screen "LLCCA_PID" 1280x800, template "Template_main"
   Button "Button_1" at 1170,125 size 106x32; TextOff 'LLCCA_PID / -'
   IOField "I/O field_4" at 220,550 size 66x32; FormatPattern 99.99; Unit  
      ProcessValue <- "LLCCA_PvSim_LLCCA_PID_DB_ioAddFactor"
   TextField "Text field_22" at 220,525 size 59x23; Text 'factor / faktor'
   IOField "I/O field_15" at 290,550 size 61x32; FormatPattern 99; Unit  s 
      ProcessValue <- "LLCCA_PvSim_LLCCA_PID_DB_ioAddTimeLag"
   TextField "Text field_23" at 290,525 size 45x23; Text 'tLag'
   Button "Button_4" at 220,680 size 156x32; TextOff 'Reset / Återställning'
      on Release: SetBit("RUN_DB_resetPvSim")
   IOField "I/O field_21" at 355,550 size 61x32; FormatPattern 999; Unit  s 
      ProcessValue <- "LLCCA_PvSim_LLCCA_PID_DB_ioAddFilter"
   TextField "Text field_25" at 355,525 size 51x23; Text 'filter'
   IOField "I/O field_22" at 220,615 size 66x32; FormatPattern 99.99; Unit  
      ProcessValue <- "LLCCA_PvSim_LLCCA_PID_DB_ioSubFactor"
   TextField "Text field_26" at 220,590 size 59x23; Text 'factor / faktor'
   IOField "I/O field_23" at 420,615 size 96x32; FormatPattern 99.9; Unit   U 
      ProcessValue <- "LLCCA_PvSim_LLCCA_PID_DB_ioSubStartValue"
   TextField "Text field_27" at 420,590 size 104x23; Text 'start value / omgivningstemp.'
   TextField "Text field_28" at 10,525 size 186x23; Text 'Additive component / Värmning'
   TextField "Text field_29" at 10,590 size 213x23; Text 'subtracting component / Kylning'
   IOField "I/O field_16" at 10,550 size 161x32; FormatPattern 999.9; Unit  U/min 
      ProcessValue <- "LLCCA_PvSim_LLCCA_PID_DB_addComp"
   IOField "I/O field_17" at 10,615 size 161x32; FormatPattern 999.9; Unit  U/min 
      ProcessValue <- "LLCCA_PvSim_LLCCA_PID_DB_subComp"
   TextField "Text field_30" at 10,655 size 66x23; Text 'Sim Pv / Simulerad temp.'
   IOField "I/O field_24" at 10,680 size 161x32; FormatPattern 999.9; Unit  U 
      ProcessValue <- "LLCCA_PvSim_LLCCA_PID_DB_out"
   TextField "Text field_31" at 10,745 size 38x23; Text 'add / värmning'
   TextField "Text field_33" at 10,765 size 36x23; Text 'sub / kylning'
   TextField "Text field_34" at 95,745 size 325x23; Text '[U/min] = factor * controller out% / [°C/min] = faktor * regulator ut%'
   TextField "Text field_35" at 95,765 size 459x23; Text '[U/min] = factor * (simulated value - start value) / [°C/min] = faktor * (simulerad temp. - omgivningstemp.)'
   TextField "Text field_32" at 5,725 size 107x23; Text 'Calculation / Hur värden beräknas'
   IOField "I/O field_6" at 380,305 size 71x32; Unit  
      ProcessValue <- "LLCCA_PID_DB_statAdvanced_derivateFilter"
   TextField "Text field_14" at 10,270 size 110x23; Text 'Parameters / Parametrar'
   IOField "I/O field_7" at 155,305 size 71x32; Unit  
      ProcessValue <- "LLCCA_PID_DB_ioKp"
   IOField "I/O field_8" at 230,305 size 71x32; Unit  
      ProcessValue <- "LLCCA_PID_DB_ioTi"
   IOField "I/O field_9" at 305,305 size 71x32; Unit  
      ProcessValue <- "LLCCA_PID_DB_ioTd"
   TextField "Text field_13" at 155,270 size 16x23; Text 'p'
   TextField "Text field_15" at 230,270 size 11x23; Text 'i'
   TextField "Text field_16" at 305,270 size 16x23; Text 'd'
   TextField "Text field_17" at 380,270 size 46x23; Text 'dFilt'
   TextField "Text field_4" at 10,40 size 53x23; Text 'Mode / Läge'
   SymbolicIOField "Symbolic I/O field_1" at 10,65 size 161x32; TextOn '1'; TextOff '0'; TextList "LLCCA_PID_state"
      ProcessValue <- "LLCCA_PID_DB_ioMode"
   IOField "I/O field_19" at 435,130 size 96x32; FormatPattern 999.9; Unit  % 
      ProcessValue <- "LLCCA_PID_DB_ManualValue"
   TextField "Text field_3" at 435,105 size 75x23; Text 'Man val / Man ut'
   IOField "I/O field_18" at 315,130 size 96x32; FormatPattern 999.9; Unit  U 
      ProcessValue <- "LLCCA_PID_DB_Setpoint"
   TextField "Text field_2" at 315,105 size 27x23; Text 'Sp / Auto sp'
   IOField "I/O field_1" at 410,680 size 96x32; FormatPattern 9.999; Unit   U 
      ProcessValue <- "LLCCA_PvSim_LLCCA_PID_DB_ioNoiceFactor"
   TextField "Text field_5" at 410,655 size 53x23; Text 'noice / omgivningstemp.'
   TextField "Text field_1" at 385,345 size 54x23; Text 'State / Läge'
   TextField "Text field_7" at 10,345 size 207x23; Text 'Method for steptuning / Method for pretuning / start up tuning'
   SymbolicIOField "Symbolic I/O field_4" at 475,370 size 361x32; TextOn '1'; TextOff '0'; TextList "LLCCA_PID_stepTuning_state"
      ProcessValue <- "LLCCA_PID_DB_statStepTuning_state"
   TextField "Text field_6" at 475,345 size 54x23; Text 'State / Läge'
   IOField "I/O field_20" at 850,370 size 96x32; FormatPattern 999; Unit  % 
      ProcessValue <- "PID_Compact_1_Progress"
   TextField "Text field_24" at 850,345 size 67x23; Text 'Tuning'
   IOField "I/O field_2" at 960,370 size 96x32; FormatPattern 999.9; Unit  s 
      ProcessValue <- "LLCCA_PID_DB_statStepTuning_t"
   TextField "Text field_8" at 960,345 size 58x23; Text 'Timer / Tuning'
   IOField "I/O field_10" at 520,615 size 96x32; FormatPattern 99.9; Unit   U 
      ProcessValue <- "LLCCA_PvSim_LLCCA_PID_DB_ioSubConstant"
   TextField "Text field_9" at 520,590 size 83x23; Text 'constant / omgivningstemp.'
   IOField "I/O field_12" at 290,615 size 61x32; FormatPattern 99; Unit  s 
      ProcessValue <- "LLCCA_PvSim_LLCCA_PID_DB_ioSubTimeLag"
   TextField "Text field_12" at 290,590 size 45x23; Text 'tLag'
   IOField "I/O field_25" at 355,615 size 61x32; FormatPattern 999; Unit  s 
      ProcessValue <- "LLCCA_PvSim_LLCCA_PID_DB_ioSubFilter"
   TextField "Text field_18" at 355,590 size 51x23; Text 'filter'
   SymbolicIOField "Symbolic I/O field_2" at 10,370 size 361x32; TextOn '1'; TextOff '0'; TextList "LLCCA_PID_stepTuning"
      ProcessValue <- "LLCCA_PID_DB_statAdvanced_tuningRule"
   IOField "I/O field_13" at 555,65 size 96x32; FormatPattern 999; Unit  U 
      ProcessValue <- "LLCCA_PID_DB_Input"
   IOField "I/O field_14" at 675,65 size 96x32; FormatPattern 999; Unit  % 
      ProcessValue <- "LLCCA_PID_DB_Out"
   TextField "Text field_10" at 555,40 size 54x23; Text 'Input / Ärvärde'
   TextField "Text field_11" at 675,40 size 67x23; Text 'Output / Utsignal'
   IOField "I/O field_27" at 555,130 size 96x32; FormatPattern 999; Unit  U 
      ProcessValue <- "LLCCA_PID_DB_Setpoint"
   TextField "Text field_21" at 555,105 size 82x23; Text 'Setpoint / Börvärde'

screen "INFO" 1280x800, template "Template_main"
   TextField "Text field_1" at 80,45 size 51x25; Text 'y(t)'
   TextField "Text field_2" at 520,350 size 31x25; Text '(t)'
   TextField "Text field_3" at 520,665 size 31x25; Text '(t)'
   TextField "Text field_4" at 515,260 size 34x25; Text 'dy'
   TextField "Text field_6" at 140,710 size 23x25; Text 'A'
   TextField "Text field_7" at 340,555 size 16x25; Text 'k'
   TextField "Text field_8" at 115,770 size 22x25; Text 'm'
   TextField "Text field_9" at 515,555 size 69x25; Text 'du = K'
   TextField "Text field_10" at 235,600 size 16x25; Text 'L'
   TextField "Text field_11" at 360,670 size 16x25; Text 'T'
   TextField "Text field_12" at 710,545 size 277x67; Text 'linear equation u = kt + m ( u=pv , t=time ) k = du / dt = u2-u1 / t2-t1'
   TextField "Text field_13" at 140,45 size 401x25; Text 'Output'
   TextField "Text field_14" at 140,360 size 401x25; Text 'Process Value = Input'
   TextField "Text field_5" at 80,360 size 51x25; Text 'u(t)'
   TextField "Text field_15" at 710,715 size 157x25; Text '1/A = T / Kp · L'
   TextField "Text field_16" at 715,100 size 267x67; Text 'TERMINOLIGY L = Lag or Deadtime T = Apparent time constant'
   TextField "Text field_17" at 715,205 size 401x235; Text 'Open-loop Ziegler-Nichols tuning method P PI 3.33L PID 2.0L 0.5L'
   TextField "Text field_18" at 780,280 size 28x25; Text 'dy'
   TextField "Text field_19" at 785,305 size 18x25; Text 'A'
   TextField "Text field_20" at 780,240 size 178x25; Text 'Kc Ti Td'
   TextField "Text field_21" at 765,340 size 58x25; Text '0.9dy'
   TextField "Text field_22" at 785,365 size 18x25; Text 'A'
   TextField "Text field_23" at 765,400 size 58x25; Text '1.2dy'
   TextField "Text field_24" at 785,425 size 18x25; Text 'A'
   Button "Button_1" at 1170,710 size 106x32; TextOff 'INFO / -'
   TextField "Text field_25" at 710,685 size 133x25; Text 'Kp = dy / du'
*)